// Mitsubishi GX Works2 project: LRI - PLC - AULA 6   PLC: Q03UDV

PROGRAM MAIN
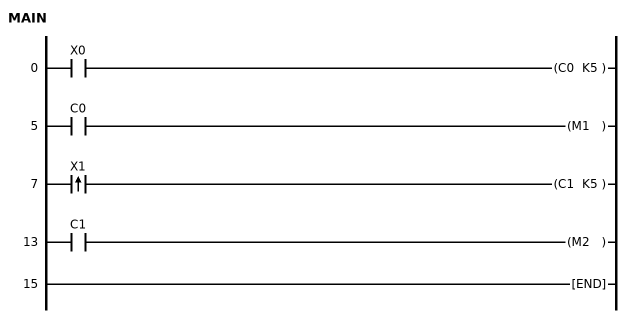
0     LD      X0
      OUT     C0 K5
5     LD      C0
      OUT     M1
7     LDP     X1
      OUT     C1 K5
13    LD      C1
      OUT     M2
15    END
END_PROGRAM
